// Virtual-commissioning application for one pneumatic press Unit.
// IMPORTANT: the Safe* values below simulate TwinSAFE outputs only. A deployed
// machine maps certified E-stop/two-hand/guard/safe-valve results from TwinSAFE.
PROGRAM MAIN
VAR
    RecipeCatalog : FB_PressRecipeCatalog;
    PartCarrier : FB_LocalPartCarrier;    // §3.16.2 BY_POSITION identity + local result ring
    AccessUsers : FB_LocalAccessProvider; // §7.7 commissioning user/PIN table
    // TF6100 TMC-Filtered publication starts at the deployed root instance.
    // The marker is inherited by PneumaticPress's published child symbols.
    {attribute 'OPC.UA.DA' := '1'}
    PneumaticPress : FB_PressDemoUnit;
    IoCatalog : FB_PressIoCatalog;
    IoDriver : FB_PressIoDriver;
    ControlDomain : FB_PressControlDomain;
    OutputAuthority : FB_PressOutputAuthority;
    SimulationDriver : FB_PressSimulationDriver;
    PressHal, DoorHal, SlideHal : ST_CylinderHal;
    TwoHandHal : ST_TwoHandHal;
    PowerHal : ST_PowerGroupHal;
    PartPresentHal : ST_DigitalInputHal;
    AirPressureHal : ST_AirPressureHal;
    HealthProbe : FB_TcSystemHealthProbe;
    HealthConfig : ST_SystemHealthParCfg;
    HealthCpuLoadPct : LREAL;
    HealthMemoryAvailableMb : UDINT;
    HealthTimeSource : STRING(32);
    InitialModel : ST_ModelId;
    Plate : ST_Nameplate;
    Init : BOOL;
    // Read-only MIRRORS of the commissioning gates (see the VAR CONSTANT block).
    // They exist only so the gate state stays visible over ADS/OPC UA: the
    // compiler inlines constants, which may publish no symbol at all, and losing
    // that visibility would remove the fastest way to diagnose "no output moves".
    // They are reassigned from the constants every cycle and nothing reads them,
    // so writing one online is inert - the constant remains the only authority.
    UseSimulation : BOOL;
    ControlCircuitMappingConfirmed : BOOL;
    // §10.5.1 demand gate, written by the HMI while its fieldbus page is open.
    // FALSE parks the EtherCAT master scan (no ADS traffic for a view nobody is
    // watching); the last read states are held, never falsified.
    FieldbusViewActive : BOOL;

    // Simulation controls. E-stop is normally closed: TRUE = healthy circuit.
    SimEStopNc : BOOL := TRUE;
    SimControlOnButton : BOOL;
    SimControlOffButton : BOOL;
    SimLeftButton : BOOL;
    SimRightButton : BOOL;
    SimSafetyValveOk : BOOL := TRUE;
    SimFieldbusHealthy : BOOL := TRUE;
    SimPartPresent : BOOL := TRUE;
    SimAirPressureOk : BOOL := TRUE;
    SafeEStopOk : BOOL;
    SafeGuardClosed : BOOL;
    SafeTwoHandActive : BOOL;
    SafePneumaticPermit : BOOL;
    SafetyFieldbusHealthy : BOOL;
    StandardIoHealthy : BOOL;
    RawEStopHealthy : BOOL;
    LampsOn : BOOL;
    ControlOnEdge : R_TRIG;
    ControlOffEdge : R_TRIG;
    ControlOnAdopted : R_TRIG;   // rising edge of the relay chain's feedback
END_VAR
VAR CONSTANT
    // COMMISSIONING GATES - deliberately CONSTANT so they cannot be flipped
    // online. Defeating a gate must be a source change plus a download: a
    // reviewable, auditable act, not a live write from an HMI or ADS client.
    //
    // TRUE makes MAIN call M_ClearOutputs() every cycle, so no physical output
    // is ever energized while the simulation driver animates the plant.
    USE_SIMULATION : BOOL := FALSE;
    // FALSE makes M_WriteOutputs force _000K951_A1 and _000K911_A1 FALSE every
    // cycle. Control On then cannot energize, the hardwired N54 D2 relay chain
    // never closes, and NOTHING moves - even though the cylinder coils are
    // written unconditionally. Set TRUE only after verifying the K951/K911
    // electrical semantics on the cabinet; per N54 D2 SwitchControlOn and
    // EnableControlOn are distinct signals.
    CONTROL_CIRCUIT_MAPPING_CONFIRMED : BOOL := TRUE;
END_VAR

// Mirror the compile-time gates so they remain observable (see declaration).
UseSimulation := USE_SIMULATION;
ControlCircuitMappingConfirmed := CONTROL_CIRCUIT_MAPPING_CONFIRMED;

IF NOT Init THEN
    Init := TRUE;
    // Initial mechanically safe/load position: ram up, door open, slide outside.
    PressHal.RetractedFb := TRUE;
    DoorHal.RetractedFb := TRUE;
    SlideHal.RetractedFb := TRUE;
    RecipeCatalog.Setup(UnitRef := PneumaticPress);
    PneumaticPress.Setup(Name := 'PneumaticPress', PressHal := PressHal, DoorHal := DoorHal,
        SlideHal := SlideHal, TwoHandHal := TwoHandHal, PowerHal := PowerHal,
        PartPresentHal := PartPresentHal, AirPressureHal := AirPressureHal,
        Recipe := RecipeCatalog.Provider);
    IoDriver.Setup(UnitRef := PneumaticPress);
    IoCatalog.Setup(UnitRef := PneumaticPress);
    ControlDomain.Setup(UnitRef := PneumaticPress);
    SimulationDriver.Setup(PressHal := PressHal, DoorHal := DoorHal, SlideHal := SlideHal);
    InitialModel.ModelCode := 'ALUMINUM';
    PneumaticPress.SetModel(Id := InitialModel);
    Plate.ProductUri := 'urn:fraktal:demo:pneumatic-press:2026-0001';
    Plate.ManufacturerName := 'Fraktal Example Project';
    Plate.ProductDesignation := 'Pneumatic Press Training Cell';
    Plate.SerialNumber := 'PRESS-DEMO-2026-0001';
    Plate.YearOfConstruction := '2026';
    Plate.SoftwareVersion := 'Fraktal Press Demo 0.1';
    PneumaticPress.SetNameplate(Plate := Plate);
    PneumaticPress.AlarmLog.RegisterMeta(Reason := E_Reason.INTERLOCK_DROPPED,
        OperatorAction := 'project.alarmAction.pressInterlock',
        Consequence := 'project.alarmConsequence.pressInterlock', Shelvable := FALSE);
    // §8.9 rationalization: per-reason operator action + consequence for the HMI join
    PneumaticPress.AlarmLog.RegisterMeta(Reason := E_Reason.PERMISSIVE_NOT_MET,
        OperatorAction := 'project.alarmAction.pressAirPressure',
        Consequence := 'project.alarmConsequence.pressAirPressure', Shelvable := FALSE);
    PneumaticPress.AlarmLog.RegisterMeta(Reason := E_Reason.RECIPE_INVALID,
        OperatorAction := 'project.alarmAction.pressRecipe',
        Consequence := 'project.alarmConsequence.pressRecipe', Shelvable := FALSE);
    PneumaticPress.AlarmLog.RegisterMeta(Reason := PL_ModuleReasons.CYL_WORK_NOT_REACHED,
        OperatorAction := 'project.alarmAction.pressCylinderPosition',
        Consequence := 'project.alarmConsequence.pressCylinderPosition', Shelvable := FALSE);
    PneumaticPress.AlarmLog.RegisterMeta(Reason := PL_ModuleReasons.CYL_HOME_NOT_REACHED,
        OperatorAction := 'project.alarmAction.pressCylinderPosition',
        Consequence := 'project.alarmConsequence.pressCylinderPosition', Shelvable := FALSE);
    // §3.16 traceability: station-local BY_POSITION serials; RFID/host substitutes later
    PartCarrier.Setup(UidPrefix := 'PRESS-2026-');
    PneumaticPress.SetPartCarrier(Carrier := PartCarrier);
    // §7.7/§14: provider secrets are retained deployment configuration, never
    // source literals. Provision them before raising any policy threshold.
    IF GVL_PressCommissioning.OperatorPin <> '' THEN
        AccessUsers.Register(User := 'operator', Pin := GVL_PressCommissioning.OperatorPin,
            Level := E_AccessLevel.OPERATOR);
    ELSE
        ;
    END_IF
    IF GVL_PressCommissioning.TechnicianPin <> '' THEN
        AccessUsers.Register(User := 'tech', Pin := GVL_PressCommissioning.TechnicianPin,
            Level := E_AccessLevel.TECHNICIAN);
    ELSE
        ;
    END_IF
    IF GVL_PressCommissioning.AdminPin <> '' THEN
        AccessUsers.Register(User := 'admin', Pin := GVL_PressCommissioning.AdminPin,
            Level := E_AccessLevel.ADMIN);
    ELSE
        ;
    END_IF
    PneumaticPress.Access.Setup(Provider := AccessUsers, pAlarmLog := ADR(PneumaticPress.AlarmLog));
    HealthConfig.MaxTaskCycleUs := 5000;
    HealthConfig.MaxTaskJitterUs := 2000;
    HealthConfig.RequireFieldbus := TRUE;
    HealthConfig.RequireDcSync := FALSE;
    HealthConfig.RequireTimeSync := TRUE;
END_IF

// Ordinary simulated local station buttons. The worksheet does not list real
// Control On/Off input buttons; physical operation therefore uses HMI requests
// until those devices are identified. Control Off wins simultaneous edges.
// Source the Control On/Off edges from the REAL buttons on a live machine, and
// from the simulated ones only under USE_SIMULATION. Previously both edges were
// ANDed with USE_SIMULATION, so on hardware neither could ever fire and the
// machine had no headless Control On path at all.
IF USE_SIMULATION THEN
    ControlOnEdge(CLK := SimControlOnButton);
    ControlOffEdge(CLK := SimControlOffButton);
ELSE
    ControlOnEdge(CLK := IoDriver.ControlOnButton);
    ControlOffEdge(CLK := IoDriver.ControlOffButton);
END_IF
IF ControlOffEdge.Q THEN
    PneumaticPress.RequestLocalControl(ControlOn := FALSE);
ELSIF ControlOnEdge.Q THEN
    PneumaticPress.RequestLocalControl(ControlOn := TRUE);
END_IF
// Adopt the relay chain's established state: it is the authority. Without this
// the PLC can sit with no power request while K911_Y32 shows control is already
// ON (observed on the press), leaving PLC and hardware permanently out of step.
// One-shot: re-issuing POWER_ON every scan would re-fault the power group on
// any momentary permit dip and spam the event log. Latch on the feedback's
// rising edge only, and re-arm the latch when control drops away.
ControlOnAdopted(CLK := PowerHal.PowerFeedback);
IF NOT USE_SIMULATION AND ControlOnAdopted.Q AND NOT ControlOffEdge.Q THEN
    PneumaticPress.RequestLocalControl(ControlOn := TRUE);
END_IF

IF USE_SIMULATION THEN
    SimulationDriver.M_ReadInputs(DoorHal := DoorHal, TwoHandHal := TwoHandHal,
        PowerHal := PowerHal, PartPresentHal := PartPresentHal,
        AirPressureHal := AirPressureHal, RawEStopHealthy := RawEStopHealthy,
        SafeEStopOk := SafeEStopOk, SafeGuardClosed := SafeGuardClosed,
        SafeTwoHandActive := SafeTwoHandActive,
        SafePneumaticPermit := SafePneumaticPermit,
        SafetyFieldbusHealthy := SafetyFieldbusHealthy,
        StandardIoHealthy := StandardIoHealthy, SimEStopNc := SimEStopNc,
        SimLeftButton := SimLeftButton, SimRightButton := SimRightButton,
        SimSafetyValveOk := SimSafetyValveOk,
        SimFieldbusHealthy := SimFieldbusHealthy,
        SimPartPresent := SimPartPresent, SimAirPressureOk := SimAirPressureOk,
        PowerRequested := PowerHal.EnableRequestOut);
ELSE
    // The project Hardware Driver is the only raw process-image consumer.
    IoDriver.M_ReadInputs(PressHal := PressHal, DoorHal := DoorHal,
        SlideHal := SlideHal, TwoHandHal := TwoHandHal, PowerHal := PowerHal,
        PartPresentHal := PartPresentHal, AirPressureHal := AirPressureHal,
        RawEStopHealthy := RawEStopHealthy, SafeEStopOk := SafeEStopOk,
        SafeGuardClosed := SafeGuardClosed, SafeTwoHandActive := SafeTwoHandActive,
        SafePneumaticPermit := SafePneumaticPermit,
        SafetyFieldbusHealthy := SafetyFieldbusHealthy,
        StandardIoHealthy := StandardIoHealthy);
END_IF
TwoHandHal.SafeActive := SafeTwoHandActive;
TwoHandHal.FieldbusHealthy := SafetyFieldbusHealthy;
PowerHal.SafetyPermit := SafePneumaticPermit;
PowerHal.FieldbusHealthy := StandardIoHealthy;

ControlDomain.M_Update(SafeEStopOk := SafeEStopOk,
    SafeGuardClosed := SafeGuardClosed, SafeTwoHandActive := SafeTwoHandActive,
    SafePneumaticPermit := SafePneumaticPermit,
    SafetyFieldbusHealthy := SafetyFieldbusHealthy,
    StandardIoHealthy := StandardIoHealthy, RawEStopHealthy := RawEStopHealthy,
    PowerFeedback := PowerHal.PowerFeedback,
    PowerRequested := PowerHal.EnableRequestOut,
    TwoHandFieldbusHealthy := TwoHandHal.FieldbusHealthy);
PneumaticPress.ControlDomain := ControlDomain.Status;

// §2.7/§8.12 framework acceptance fixture. Simulation supplies explicit healthy
// synthetic controller/time probes; a real target stays conspicuously
// unavailable until its platform metrics and documented sync source are wired.
IF USE_SIMULATION THEN
    HealthCpuLoadPct := 25.0;
    HealthMemoryAvailableMb := UDINT#1024;
    HealthTimeSource := 'SIMULATED';
ELSE
    HealthCpuLoadPct := 0.0;
    HealthMemoryAvailableMb := UDINT#0;
    HealthTimeSource := 'UNCONFIGURED';
END_IF
HealthProbe.Cyclic(ExpectedCycleUs := 1000, ExternalTaskOverrun := FALSE,
    ControllerAvailable := USE_SIMULATION,
    CpuLoadPct := HealthCpuLoadPct,
    MemoryAvailableMb := HealthMemoryAvailableMb,
    IpcAvailable := FALSE, IpcTemperatureC := 0.0,
    FanHealthy := TRUE, StorageHealthPct := 100.0,
    FieldbusAvailable := TRUE, FieldbusMasterHealthy := StandardIoHealthy,
    LostFrameCount := 0, SlaveErrorCount := 0,
    DcAvailable := USE_SIMULATION, DcSynchronized := USE_SIMULATION,
    TimeAvailable := USE_SIMULATION, TimeSynchronized := USE_SIMULATION,
    TimeSource := HealthTimeSource,
    TimeOffsetUs := 0, LastSyncAt := F_Now());
IF HealthProbe.Health.TaskAvailable THEN
    PneumaticPress.SetSystemHealth(Input := HealthProbe.Health, ParCfg := HealthConfig);
ELSE
    ; // first monotonic sample has no prior scan from which to derive a period
END_IF

// First execute ordinary control, then apply a standard-PLC withdrawal layer.
// This is defense in depth only: the real safety system owns pneumatic removal.
PneumaticPress();
OutputAuthority.M_Apply(PressHal := PressHal, DoorHal := DoorHal,
    SlideHal := SlideHal, PowerFeedback := PowerHal.PowerFeedback,
    SafePneumaticPermit := SafePneumaticPermit,
    StandardIoHealthy := StandardIoHealthy,
    HazardousRamPermit := SafeGuardClosed AND SafeTwoHandActive);
IF USE_SIMULATION THEN
    // Never leave physical outputs energized while virtual commissioning.
    IoDriver.M_ClearOutputs();
    SimulationDriver.M_RefreshPlant();
ELSE
    LampsOn := PneumaticPress.TwoHand.OutImm.Armed
        AND ControlDomain.Status.ReadyForStart
        AND PneumaticPress.OutImm.PartPresent AND PneumaticPress.OutImm.AirPressureOk;
    IoDriver.M_WriteOutputs(PressHal := PressHal, DoorHal := DoorHal,
        SlideHal := SlideHal, PowerHal := PowerHal, LampsOn := LampsOn,
        ControlCircuitMappingConfirmed := CONTROL_CIRCUIT_MAPPING_CONFIRMED);
END_IF
// Node state comes from the real EtherCAT master. §10.5.1 is a diagnostic
// surface, so the master is scanned only while a client is watching the bus
// view: the HMI sets FieldbusViewActive when its fieldbus page is open (the same
// on-demand gating the read tiers already apply to the topology data itself).
IoDriver.M_RefreshFieldbus(BusViewActive := FieldbusViewActive);

END_PROGRAM

(* stored: Version 1.1.0.1, ProductVersion 3.1.4024.16
   POU MAIN: Id {55a765e4-afc1-4fdb-91af-a60d34c2c143}, SpecialFunc None *)
